{attribute 'qualified_only'}
VAR_GLOBAL
	T1				AT %I*	: BOOL; 
	T2				AT %I*	: BOOL; 
	P				AT %I*	: INT; 	
	LED_Green 		AT %Q* : BOOL;
	LED_Yellow 		AT %Q* : BOOL;
	LED_Red 		AT %Q* : BOOL;
END_VAR

(* stored: Version 1.1.0.1
   GVL IO_PLC: Id {d2f65eac-ad92-41eb-ad1f-127351d08df8} *)
